Staubli VAL3: encode.pgx

public program encode(num& x_nStatus (dimensions=1), num& x_nOutputBuffer[] (dimensions=1))
  local num l_nDWordBytes[4]
  local num l_nBufferPos
  local num i
begin
  if x_nStatus<0
    return
  endIf
  l_nBufferPos=0
  x_nStatus=0
  call encodeSharedInt(x_nStatus,x_nOutputBuffer,l_nBufferPos,prefix.nLength)
  call encodeSharedInt(x_nStatus,x_nOutputBuffer,l_nBufferPos,header.nMsgType)
  call encodeSharedInt(x_nStatus,x_nOutputBuffer,l_nBufferPos,header.nCommType)
  call encodeSharedInt(x_nStatus,x_nOutputBuffer,l_nBufferPos,header.nReplyCode)
  call encodeSharedInt(x_nStatus,x_nOutputBuffer,l_nBufferPos,body.robotId)
  call encodeSharedInt(x_nStatus,x_nOutputBuffer,l_nBufferPos,body.sequence)
  call encodeSharedInt(x_nStatus,x_nOutputBuffer,l_nBufferPos,body.validFields)
  call encodeShareReal(x_nStatus,x_nOutputBuffer,l_nBufferPos,body.time)
  call encodeJointData(x_nStatus,x_nOutputBuffer,l_nBufferPos,body.positions)
  call encodeJointData(x_nStatus,x_nOutputBuffer,l_nBufferPos,body.velocities)
  call encodeJointData(x_nStatus,x_nOutputBuffer,l_nBufferPos,body.accelerations)
end
